FUNCTION_BLOCK FB_Vending
VAR_INPUT
END_VAR
VAR_OUTPUT
END_VAR
VAR
	coinsinsert : REAL;
	{attribute 'OPC.UA.DA' :='1'}
	Logistic : LogStruct;
	{attribute 'OPC.UA.DA' :='1'}
	stock : ARRAY[0..8] OF INT := [3, 3, 3, 3, 3, 3, 3, 3, 3];

	ncase: INT; 
	timer: ARRAY[1..3] OF TON;
	i : INT;
	
	tim : TON;
	osTim : TON;
	O: INT;
	MoveAxis1 : MC_MoveAbsolute;
	Reset : MC_Reset;
	Power : Tc2_MC2.MC_Power;
END_VAR

GVL.Axis1.ReadStatus(); 

IF GVL.potentiometer1 < 0 THEN
	coinsinsert := 0;
ELSE
	coinsinsert := (INT_TO_REAL(GVL.potentiometer1)/32767)*10; 
END_IF
// scalling potentiometer 1-10

CASE ncase OF
0:
MoveAxis1.Execute:=FALSE;
Reset.Execute:=FALSE; 
Power.Enable:=TRUE; 
Power.Enable_Positive:=TRUE; 
Power.Enable_Negative:=TRUE; 
ncase:= 60;

10:
IF GVL.button1 THEN
	GVL.number:= '1';
	ncase:= 20;
ELSIF GVL.button2 THEN
	GVL.number:= '2';
	ncase:= 20;
ELSIF GVL.button3 THEN
	GVL.number:= '3';
	ncase:= 20;
ELSIF GVL.buttonA THEN
	GVL.letter:= 'A';
	ncase:= 30;
ELSIF GVL.buttonB THEN
	GVL.letter:= 'B';
	ncase:= 30;
ELSIF GVL.buttonC THEN
	GVL.letter:= 'C';
	ncase:= 30;
END_IF

20:
IF GVL.button1 THEN
	GVL.number:= '1';
	ncase:= 20;
ELSIF GVL.button2 THEN
	GVL.number:= '2';
	ncase:= 20;
ELSIF GVL.button3 THEN
	GVL.number:= '3';
	ncase:= 20;
ELSIF GVL.buttonA THEN
	GVL.letter:= 'A';
	ncase:= 40;
ELSIF GVL.buttonB THEN
	GVL.letter:= 'B';
	ncase:= 40;
ELSIF GVL.buttonC THEN
	GVL.letter:= 'C';	
	ncase:= 40;
END_IF

30:
IF GVL.button1 THEN
	GVL.number:= '1';
	ncase:= 40;
ELSIF GVL.button2 THEN
	GVL.number:= '2';
	ncase:= 40;
ELSIF GVL.button3 THEN
	GVL.number:= '3';
	ncase:= 40;
ELSIF GVL.buttonA THEN
	GVL.letter:= 'A';
	ncase:= 30;
ELSIF GVL.buttonB THEN
	GVL.letter:= 'B';
	ncase:= 30;
ELSIF GVL.buttonC THEN
	GVL.letter:= 'C';
	ncase:= 30;
END_IF

40:
	IF GVL.buttonO THEN
		IF GVL.number = '1' AND GVL.letter = 'A' AND coinsinsert >= 1.6 THEN
			IF stock[0] =0 THEN 
				GVL.dcoins := coinsinsert; 
				GVL.osled[0] := TRUE;
				GVL.led1 := TRUE;
				GVL.sufficiency:= 'NO STOCK';
				osTim(IN := TRUE, PT :=T#5S);
				IF osTim.Q THEN
					osTim(IN := FALSE);
					ncase := 60;
				END_IF
			ELSE
				GVL.dcoins := coinsinsert;
				GVL.led[1]:= TRUE;	// DISPENSE ITEM LAMP ON
				GVL.osled[0] := FALSE; // OUT OF STOCK LAMP OFF
				GVL.xvar[1]:= 0;
				GVL.yvar[1]:= 0;
				GVL.change:= coinsinsert - 1.6;
				Logistic.sales := Logistic.sales + 1.6;
				GVL.sufficiency:= 'Thank You';
				ncase:= 80;
				i := 0;
			
			END_IF
		
		ELSIF GVL.number = '1' AND GVL.letter = 'B' AND coinsinsert >= 1.90 THEN
			IF stock[1] =0 THEN
					GVL.dcoins := coinsinsert; 
					GVL.osled[1] := TRUE;
					GVL.sufficiency:= 'NO STOCK';
					osTim(IN := TRUE, PT :=T#5S);
				IF osTim.Q THEN
					osTim(IN := FALSE);
					ncase := 60;
				END_IF
			ELSE
				GVL.dcoins := coinsinsert;
				GVL.led[2]:= TRUE;			// DISPENSE ITEM
				GVL.osled[1] := FALSE;		// OUT OF STOCK LAMP OFF
				GVL.xvar[2]:= 0;					
				GVL.yvar[2]:= 0;
				GVL.change:= coinsinsert - 1.9;
				Logistic.sales := Logistic.sales + 1.9;
				GVL.sufficiency:= 'Thank You';
				ncase:= 80;
				i := 1;
			END_IF
				
		ELSIF GVL.number='1' AND GVL.letter='C' AND coinsinsert >=2 THEN
			IF stock[2] =0 THEN 
					GVL.dcoins := coinsinsert;
					GVL.osled[2] := TRUE;
					GVL.sufficiency:= 'NO STOCK';
					osTim(IN := TRUE, PT :=T#5S);
				IF osTim.Q THEN
					osTim(IN := FALSE);
					ncase := 60;
				END_IF
			ELSE
				GVL.dcoins := coinsinsert;
				GVL.led[3]:= TRUE;			// DISPENSE ITEM        
				GVL.osled[2] := FALSE;      // OUT OF STOCK LAMP OFF
				GVL.xvar[3]:= 0;
				GVL.yvar[3]:= 0;		
				GVL.change:= coinsinsert - 2;
				Logistic.sales := Logistic.sales + 2;
				GVL.sufficiency:= 'Thank You';
				ncase:= 80;
				i := 2;
				
			END_IF
			
		ELSIF GVL.number = '2' AND GVL.letter = 'A' AND coinsinsert >= 1.6 THEN
			IF stock[3] =0 THEN 
					GVL.dcoins := coinsinsert;
					GVL.osled[3] := TRUE;
					GVL.sufficiency:= 'NO STOCK';
					osTim(IN := TRUE, PT :=T#5S);
				IF osTim.Q THEN
					osTim(IN := FALSE);
					ncase := 60;
				END_IF
			ELSE
				GVL.dcoins := coinsinsert;
				GVL.led[4]:= TRUE;
				GVL.osled[3] := FALSE;
				GVL.xvar[4]:= 0;
				GVL.yvar[4]:= 0;
				GVL.change:= coinsinsert - 1.6;
				Logistic.sales := Logistic.sales + 1.6;
				GVL.sufficiency:= 'Thank You';
				ncase:= 80;
				i := 3;
			END_IF
			
			ELSIF GVL.number = '2' AND GVL.letter = 'B' AND coinsinsert >= 1.4 THEN
				IF stock[4] =0 THEN
					GVL.dcoins := coinsinsert; 
					GVL.osled[4] := TRUE;
					GVL.sufficiency:= 'NO STOCK';
					osTim(IN := TRUE, PT :=T#5S);
				IF osTim.Q THEN
					osTim(IN := FALSE);
					ncase := 60;
				END_IF
			ELSE
				GVL.dcoins := coinsinsert;
				GVL.led[5]:= TRUE;
				GVL.osled[4] := FALSE;
				GVL.xvar[5]:= 0;
				GVL.yvar[5]:= 0;
				GVL.change:= coinsinsert - 1.4;
				Logistic.sales := Logistic.sales + 1.4;
				GVL.sufficiency:= 'Thank You';
				ncase:= 80;
				i := 4;
			END_IF
			
			ELSIF GVL.number = '2' AND GVL.letter = 'C' AND coinsinsert >= 0.8 THEN
				IF stock[5] =0 THEN
					GVL.dcoins := coinsinsert; 
					GVL.sufficiency:= 'NO STOCK';
					osTim(IN := TRUE, PT :=T#5S);
				IF osTim.Q THEN
					osTim(IN := FALSE);
					ncase := 60;
				END_IF
			ELSE
				GVL.dcoins := coinsinsert;
				GVL.led[6]:= TRUE;
				GVL.osled[5] := FALSE;
				GVL.xvar[6]:= 0;
				GVL.yvar[6]:= 0;
				GVL.change:= coinsinsert - 0.8;
				Logistic.sales := Logistic.sales + 0.8;
				GVL.sufficiency:= 'Thank You';
				ncase:= 80;
				i := 5;
			END_IF
			
			ELSIF GVL.number = '3' AND GVL.letter = 'A' AND coinsinsert >= 1.3 THEN
				IF stock[6] =0 THEN
					GVL.dcoins := coinsinsert;
					GVL.osled[6] := TRUE; 
					GVL.sufficiency:= 'NO STOCK';
					osTim(IN := TRUE, PT :=T#5S);
				IF osTim.Q THEN
					osTim(IN := FALSE);
					ncase := 60;
				END_IF
			ELSE
				GVL.dcoins := coinsinsert;
				GVL.led[7]:= TRUE;
				GVL.osled[6] := FALSE;
				GVL.xvar[7]:= 0;
				GVL.yvar[7]:= 0;
				GVL.change:= coinsinsert - 1.3;
				Logistic.sales := Logistic.sales + 1.3;
				GVL.sufficiency:= 'Thank You';
				ncase:= 80;
				i := 6;
			END_IF
			
			ELSIF GVL.number = '3' AND GVL.letter = 'B' AND coinsinsert >= 1.3 THEN
				IF stock[7] =0 THEN
					GVL.dcoins := coinsinsert;
					GVL.osled[7] := TRUE; 
					GVL.sufficiency:= 'NO STOCK';
					osTim(IN := TRUE, PT :=T#5S);
				IF osTim.Q THEN
					osTim(IN := FALSE);
					ncase := 60;
				END_IF
			ELSE
				GVL.dcoins := coinsinsert;
				GVL.led[8]:= TRUE;
				GVL.osled[7] := FALSE;
				GVL.xvar[8]:= 0;
				GVL.yvar[8]:= 0;
				GVL.change:= coinsinsert - 1.3;
				Logistic.sales := Logistic.sales + 1.3;
				GVL.sufficiency:= 'Thank You';
				ncase:= 80;
				i := 7;
			END_IF
			
			ELSIF GVL.number = '3' AND GVL.letter = 'C' AND coinsinsert >= 1.5 THEN
				IF stock[8] =0 THEN
					GVL.dcoins := coinsinsert;
					GVL.osled[8] := TRUE; 
					GVL.sufficiency:= 'NO STOCK';
					osTim(IN := TRUE, PT :=T#5S);
				IF osTim.Q THEN
					osTim(IN := FALSE);
					ncase := 60;
				END_IF
			ELSE
				GVL.dcoins := coinsinsert;
				GVL.led[9]:= TRUE;
				GVL.osled[8] := FALSE;
				GVL.xvar[9]:= 0;
				GVL.yvar[9]:= 0;
				GVL.change:= coinsinsert - 1.5;
				Logistic.sales := Logistic.sales + 1.5;
				GVL.sufficiency:= 'Thank You';
				ncase:= 80;
				i := 8;
			END_IF
			
	ELSE
		GVL.sufficiency:= 'Insufficient';
		ncase:= 70; 
END_IF
	

END_IF



50:
MoveAxis1.Position:=0; 
MoveAxis1.Velocity:=1000;     
MoveAxis1.Execute:=TRUE; 
stock[i] := stock[i] -1;

ncase:= 100;

60:
GVL.buttonO:= FALSE;
GVL.dcoins:= 0;
GVL.dchange:= 0;
GVL.number:= ' ';
GVL.letter:= ' ';
GVL.sufficiency:= ' ';
GVL.xvar[1]:= 300;
GVL.yvar[1]:= 400;
GVL.xvar[2]:= 300;
GVL.yvar[2]:= 400;
GVL.xvar[3]:= 300;
GVL.yvar[3]:= 400;
GVL.xvar[4]:= 300;
GVL.yvar[4]:= 400;
GVL.xvar[5]:= 300;
GVL.yvar[5]:= 400;
GVL.xvar[6]:= 300;
GVL.yvar[6]:= 400;
GVL.xvar[7]:= 300;
GVL.yvar[7]:= 400;
GVL.xvar[8]:= 300;
GVL.yvar[8]:= 400;
GVL.xvar[9]:= 300;
GVL.yvar[9]:= 400;
GVL.led[1]:= FALSE;
GVL.led[2]:= FALSE;
GVL.led[3]:= FALSE;
GVL.led[4]:= FALSE;
GVL.led[5]:= FALSE;
GVL.led[6]:= FALSE;
GVL.led[7]:= FALSE;
GVL.led[8]:= FALSE;
GVL.led[9]:= FALSE;
ncase:= 10;

70:
tim(IN := TRUE, PT :=T#5S);
IF tim.Q THEN
	tim(IN := FALSE);
	ncase:= 71;
END_IF

71:
IF stock[0] = 0 THEN
	GVL.osled[0] := TRUE;
	ncase:= 72;
ELSE
	ncase := 72;
	
	END_IF
	
72:
IF stock[1] = 0 THEN
	GVL.osled[1] := TRUE;
	ncase:= 73;
	ELSE
	ncase := 73;
	END_IF
73:
IF stock[2] = 0 THEN
	GVL.osled[2] := TRUE;
	ncase:= 74;
	ELSE
	ncase := 74;
	END_IF
74:
IF
	stock[3] = 0 THEN
	GVL.osled[3] := TRUE;
	ncase:= 75;
	ELSE
	ncase := 75;
	END_IF
75:
IF
	stock[4] = 0 THEN
	GVL.osled[4] := TRUE;
	ncase:= 76;
	ELSE
	ncase := 76;
	END_IF
76:
IF
	stock[5] = 0 THEN
	GVL.osled[5] := TRUE;
	ncase:= 77;
	ELSE
	ncase := 77;
	END_IF
77:
IF
	stock[6] = 0 THEN
	GVL.osled[6] := TRUE;
	ncase:= 78;
	ELSE
	ncase := 78;
	END_IF
78:
IF stock[7] = 0 THEN
	GVL.osled[7] := TRUE;
	ncase:= 79;
	ELSE
	ncase := 79;
	END_IF
79:	
IF stock[8] = 0 THEN
	GVL.osled[8] := TRUE;
	ncase:= 60;
	ELSE
	ncase := 60;

END_IF

80:
MoveAxis1.Position:=2000; 
MoveAxis1.Velocity:=1000;     
MoveAxis1.Execute:=TRUE;    
IF MoveAxis1.Done THEN  
	MoveAxis1.Execute:=FALSE; 
	GVL.buttonO:= FALSE;
	ncase:= 90;
END_IF

90:
timer[1](IN:= TRUE, PT:= T#0.5S);
IF timer[1].Q THEN
	timer[1](IN:= FALSE);
	ncase:= 50;
END_IF

100:
IF MoveAxis1.Done THEN  
	MoveAxis1.Execute:=FALSE; 
	GVL.dcoins := coinsinsert;
	GVL.dchange:= GVL.change;
	
	ncase:= 70; 
END_IF



END_CASE
ActPower();  
ActMove(); 
ActReset();

ACTION ActMove:
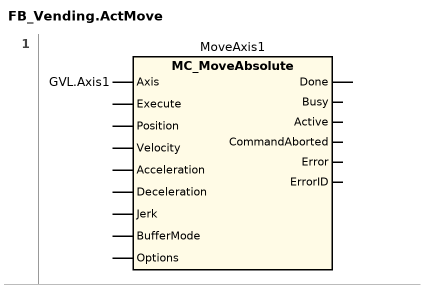
// NETWORK 1
MoveAxis1(Axis := GVL.Axis1); // MC_MoveAbsolute
END_ACTION

ACTION ActPower:
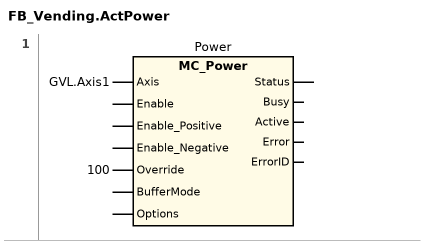
// NETWORK 1
Power(Axis := GVL.Axis1, Override := 100); // MC_Power
END_ACTION

ACTION ActReset:
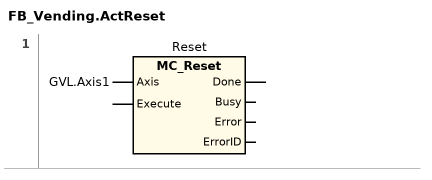
// NETWORK 1
Reset(Axis := GVL.Axis1); // MC_Reset
END_ACTION

END_FUNCTION_BLOCK

(* stored: Version 1.1.0.1, ProductVersion 3.1.4024.10
   POU FB_Vending: Id {ecbe2eca-4327-46a6-a96d-0332673f8ed6}, SpecialFunc None
   Action ActMove: Id {5d9af8c5-5509-407f-bc44-35e4328c501f}
   Action ActPower: Id {809b70a2-6505-4f08-a220-a126e5fe51f8}
   Action ActReset: Id {8bfa41bd-a4d0-4251-b262-15d363adbdd2} *)
